PROGRAM MAIN
VAR
	//Axis
	positionDrive: FB_MOVIKITpositioningDrive;
	stDrive: stMOVIKITpositioningDrive;
	
	//Logic
	_uiState			: UINT;
END_VAR

//Beispiel Aufruf mit zentraler Struktur als Referenz übergeben
//positionDrive(example_stMovikitpositioningDrive := positionDriveStruct);

MotorMovementStateMachine();

MapStructureToMovicKitFB();

ACTION MapStructureToMovicKitFB:
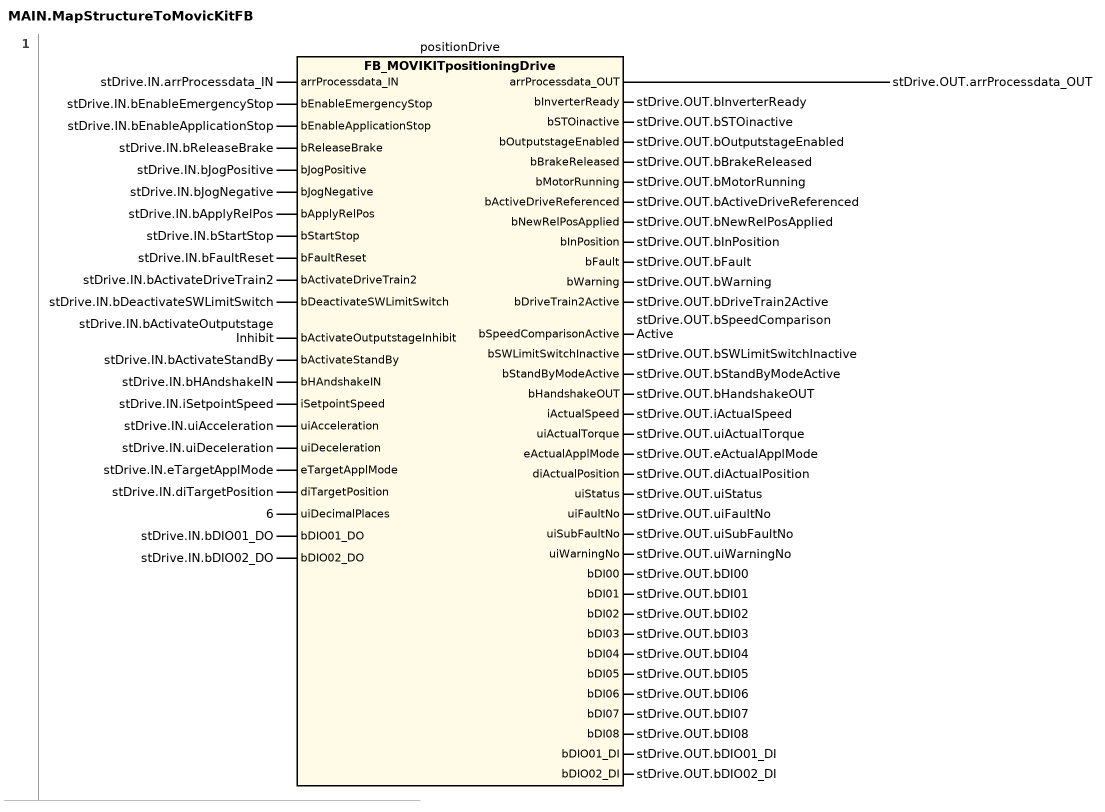
// NETWORK 1
positionDrive(
    arrProcessdata_IN := stDrive.IN.arrProcessdata_IN,
    bEnableEmergencyStop := stDrive.IN.bEnableEmergencyStop,
    bEnableApplicationStop := stDrive.IN.bEnableApplicationStop,
    bReleaseBrake := stDrive.IN.bReleaseBrake,
    bJogPositive := stDrive.IN.bJogPositive,
    bJogNegative := stDrive.IN.bJogNegative,
    bApplyRelPos := stDrive.IN.bApplyRelPos,
    bStartStop := stDrive.IN.bStartStop,
    bFaultReset := stDrive.IN.bFaultReset,
    bActivateDriveTrain2 := stDrive.IN.bActivateDriveTrain2,
    bDeactivateSWLimitSwitch := stDrive.IN.bDeactivateSWLimitSwitch,
    bActivateOutputstageInhibit := stDrive.IN.bActivateOutputstageInhibit,
    bActivateStandBy := stDrive.IN.bActivateStandBy,
    bHAndshakeIN := stDrive.IN.bHAndshakeIN,
    iSetpointSpeed := stDrive.IN.iSetpointSpeed,
    uiAcceleration := stDrive.IN.uiAcceleration,
    uiDeceleration := stDrive.IN.uiDeceleration,
    eTargetApplMode := stDrive.IN.eTargetApplMode,
    diTargetPosition := stDrive.IN.diTargetPosition,
    uiDecimalPlaces := 6,
    bDIO01_DO := stDrive.IN.bDIO01_DO,
    bDIO02_DO := stDrive.IN.bDIO02_DO,
    bInverterReady => stDrive.OUT.bInverterReady,
    bSTOinactive => stDrive.OUT.bSTOinactive,
    bOutputstageEnabled => stDrive.OUT.bOutputstageEnabled,
    bBrakeReleased => stDrive.OUT.bBrakeReleased,
    bMotorRunning => stDrive.OUT.bMotorRunning,
    bActiveDriveReferenced => stDrive.OUT.bActiveDriveReferenced,
    bNewRelPosApplied => stDrive.OUT.bNewRelPosApplied,
    bInPosition => stDrive.OUT.bInPosition,
    bFault => stDrive.OUT.bFault,
    bWarning => stDrive.OUT.bWarning,
    bDriveTrain2Active => stDrive.OUT.bDriveTrain2Active,
    bSpeedComparisonActive => stDrive.OUT.bSpeedComparisonActive,
    bSWLimitSwitchInactive => stDrive.OUT.bSWLimitSwitchInactive,
    bStandByModeActive => stDrive.OUT.bStandByModeActive,
    bHandshakeOUT => stDrive.OUT.bHandshakeOUT,
    iActualSpeed => stDrive.OUT.iActualSpeed,
    uiActualTorque => stDrive.OUT.uiActualTorque,
    eActualApplMode => stDrive.OUT.eActualApplMode,
    diActualPosition => stDrive.OUT.diActualPosition,
    uiStatus => stDrive.OUT.uiStatus,
    uiFaultNo => stDrive.OUT.uiFaultNo,
    uiSubFaultNo => stDrive.OUT.uiSubFaultNo,
    uiWarningNo => stDrive.OUT.uiWarningNo,
    bDI00 => stDrive.OUT.bDI00,
    bDI01 => stDrive.OUT.bDI01,
    bDI02 => stDrive.OUT.bDI02,
    bDI03 => stDrive.OUT.bDI03,
    bDI04 => stDrive.OUT.bDI04,
    bDI05 => stDrive.OUT.bDI05,
    bDI06 => stDrive.OUT.bDI06,
    bDI07 => stDrive.OUT.bDI07,
    bDI08 => stDrive.OUT.bDI08,
    bDIO01_DI => stDrive.OUT.bDIO01_DI,
    bDIO02_DI => stDrive.OUT.bDIO02_DI); // FB_MOVIKITpositioningDrive
stDrive.OUT.arrProcessdata_OUT := positionDrive.arrProcessdata_OUT;
END_ACTION

ACTION MotorMovementStateMachine:
CASE _uiState OF
	
	//Initialisieren
	0:
		IF NOT stDrive.Out.bFault THEN
			_uiState := 0;
		END_IF

	//Generiere Fahrbefehl auf 0mm
	10:
		stDrive.IN.eTargetApplMode			:= eMOVIKITpositioningDrive_ApplMode.PositionAbs;
		stDrive.IN.bEnableApplicationStop	:= TRUE;		//TRUE = Freigabe
		stDrive.IN.bEnableEmergencyStop		:= TRUE;		//TRUE = Freigabe
		stDrive.IN.uiAcceleration			:= 100;			//[Anwendereinheit in der Achse]
		stDrive.IN.uiDeceleration			:= 100;			//[Anwendereinheit in der Achse]
		stDrive.IN.iSetpointSpeed			:= 30;			//[Anwendereinheit in der Achse]
		stDrive.IN.diTargetPosition			:= 0;			//[Anwendereinheit in der Achse]
		stDrive.IN.bStartStop				:= TRUE;		//TRUE = Freigabe Positionierbefehl
		_uiState := 20;
		
		
		
	//Warte auf Achse in Position
	20:
		//Varianten für In pos abfragen
		//1. zeitverzögert fragen
		//2. Istposition abgleichen mit Sollposition
			IF ABS(stDrive.OUT.diActualPosition - stDrive.IN.diTargetPosition) < 1 THEN
				_uiState := 30;
			END_IF
	

	30:
	//Generiere Fahrbefehl auf 1000mm
		stDrive.IN.eTargetApplMode			:= eMOVIKITpositioningDrive_ApplMode.PositionAbs;
		stDrive.IN.bEnableApplicationStop	:= TRUE;		//TRUE = Freigabe
		stDrive.IN.bEnableEmergencyStop		:= TRUE;		//TRUE = Freigabe
		stDrive.IN.uiAcceleration			:= 100;			//[Anwendereinheit in der Achse]
		stDrive.IN.uiDeceleration			:= 100;			//[Anwendereinheit in der Achse]
		stDrive.IN.iSetpointSpeed			:= 30;			//[Anwendereinheit in der Achse]
		stDrive.IN.diTargetPosition			:= 1000;		//[Anwendereinheit in der Achse]
		stDrive.IN.bStartStop				:= TRUE;		//TRUE = Freigabe Positionierbefehl
		_uiState := 35;	

		
	35:
		//Warte auf Achse in Position
		//Varianten für In pos abfragen
		//1. zeitverzögert fragen
		//2. Istposition abgleichen mit Sollposition
			IF ABS(stDrive.OUT.diActualPosition - stDrive.IN.diTargetPosition) < 1 THEN
				_uiState := 10;
			END_IF	
	
	
	//Antrieb stoppen
	40:
		//Variante 1: Antrieb verbleibt in Lageregelung (Motor bestromt)
		stDrive.IN.bStartStop				:= FALSE;		//TRUE = Freigabe Positionierbefehl
		
		//Variante 2: Antrieb lässt Bremse einfallen und beendet Bestromung
		stDrive.IN.bEnableApplicationStop	:= FALSE;		//TRUE = Freigabe
		
	45: 
		stDrive.In.eTargetApplMode			:= eMOVIKITpositioningDrive_ApplMode.ReferenceOffsFieldb;
		stDrive.IN.bEnableEmergencyStop		:= TRUE;		//TRUE = Freigabe
		stDrive.IN.bEnableApplicationStop	:= TRUE;		//TRUE = Freigabe
		stDrive.IN.bStartStop				:= TRUE;		//TRUE = Freigabe Positionierbefehl
		//IF stDrive.OUT.bActiveDriveReferenced = TRUE THEN
		//	_uiState := 0;
		//END_IF
		
	50: 
		stDrive.IN.bFaultReset := TRUE; 
		IF stDrive.OUT.bFault = FALSE THEN 
			stDrive.IN.bFaultReset := FALSE; 
			_uiState := 0; 
		END_IF
		
	60:
	//Generiere Fahrbefehl auf 1000mm
		stDrive.IN.eTargetApplMode			:= eMOVIKITpositioningDrive_ApplMode.PositionAbs;
		stDrive.IN.bEnableApplicationStop	:= TRUE;		//TRUE = Freigabe
		stDrive.IN.bEnableEmergencyStop		:= TRUE;		//TRUE = Freigabe
		stDrive.IN.uiAcceleration			:= 100;			//[Anwendereinheit in der Achse]
		stDrive.IN.uiDeceleration			:= 100;			//[Anwendereinheit in der Achse]
		stDrive.IN.iSetpointSpeed			:= 30;			//[Anwendereinheit in der Achse]
		stDrive.IN.diTargetPosition			:= -45280;		//[Anwendereinheit in der Achse]
		stDrive.IN.bStartStop				:= TRUE;		//TRUE = Freigabe Positionierbefehl
		_uiState := 0;	


END_CASE
END_ACTION

END_PROGRAM

(* stored: Version 1.1.0.1, ProductVersion 3.1.4024.11
   POU MAIN: Id {e8daf5db-9001-4d7d-a93e-b77cf75fbe13}, SpecialFunc None
   Action MapStructureToMovicKitFB: Id {9b3e020e-43e5-4b1e-9b84-345144a7e5f1}
   Action MotorMovementStateMachine: Id {0331d407-d3a0-4019-baa4-858cca224f21} *)
